TYPE PuckTrack_typ :
STRUCT

	PuckPresent			: BOOL;
	ConveyorPosition	: LREAL;
	YPosition			: LREAL;

END_STRUCT
END_TYPE

(* stored: Version 1.1.0.1, ProductVersion 3.1.4024.9
   DUT PuckTrack_typ: Id {792a6d78-119e-4b4e-9266-cc50b03becc5} *)
